SUBAPPLICATION Uebung_007d_AX (* Blinker mit E_CYCLE und E_T_FF *)
  (* Standard: 61499-2; Description: Copyright (c) 2023 Meisterschulen am Ostbahnhof This program and the accompanying materials are made available under the terms of the Eclipse Public License 2.0 which is available at https://www.eclipse.org/legal/epl-2.0/ SPDX-License-Identifier: EPL-2.0 *)
  (* Version 1.0, 2023-10-23, Franz Höpfinger, Meisterschulen am Ostbahnhof, initial API and implementation and/or initial documentation *)
  PACKAGE Uebungen;
  IMPORT logiBUS::io::DQ::logiBUS_DO::Output_Q1;
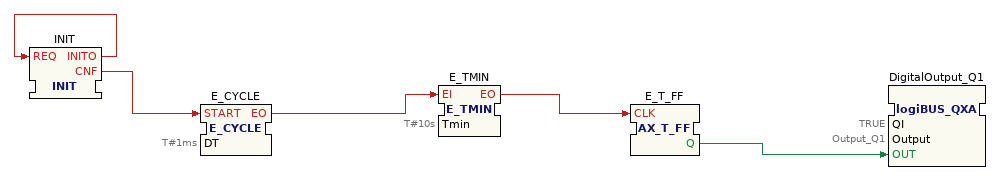
  FBS
    DigitalOutput_Q1 : logiBUS::io::DQ::logiBUS_QXA(QI := TRUE, Output := Output_Q1);
    E_CYCLE : iec61499::events::E_CYCLE(DT := T#1ms);
    E_T_FF : adapter::events::unidirectional::AX_T_FF;
    E_TMIN : iec61499::events::E_TMIN(Tmin := T#10s);
    INIT : iec61131::booleanOperators::INIT;
  END_FBS
  EVENT_CONNECTIONS
    E_CYCLE.EO TO E_TMIN.EI;
    E_TMIN.EO TO E_T_FF.CLK;
    INIT.INITO TO INIT.REQ;
    INIT.CNF TO E_CYCLE.START;
  END_CONNECTIONS
  ADAPTER_CONNECTIONS
    E_T_FF.Q TO DigitalOutput_Q1.OUT;
  END_CONNECTIONS
END_SUBAPPLICATION
